!
!1606R04_1606R06
KOLLISION_ZONE 6\Anfrage;
!
!1606R04_1606R06
KOLLISION_ZONE 7\Anfrage;
!
!1606R04_1606R06
KOLLISION_ZONE 8\Anfrage;
!
MoveJ LHP_600, vSchnell, fine, nomtcp1\WObj:=BS_1606_1A;
!
!1606R04_1606R06
KOLLISION_ZONE 1\Anfrage;
!
MoveJ LHP_005,vSchnell,z100,nomtcp1\WObj:=BS_1606_1A;
MoveJ LHP_010,vSchnell,z100,nomtcp1\WObj:=BS_1606_1A;
MoveJ LHP_015,vSchnell,z100,nomtcp1\WObj:=BS_1606_1A;
MoveJ LHP_020,vSchnell,z100,nomtcp1\WObj:=BS_1606_1A;
MoveJ LHP_025,vSchnell,z100,nomtcp1\WObj:=BS_1606_1A;
MoveJ LHP_030,vSchnell,z100,nomtcp1\WObj:=BS_1606_1A;
MoveJ LHP_035, vSchnell, z100, nomtcp1\WObj:=BS_1606_1A;
!
SpotL G0216023682BP20\VFO:=210,vSpot,nomtcp1\WObj:=BS_1606_1A;
!
MoveJ LHP_040,vSchnell,z100,nomtcp1\WObj:=BS_1606_1A;
!
SpotL G0216190516BP20\VFO:=210,vSpot,nomtcp1\WObj:=BS_1606_1A;
!
MoveJ LHP_045,vSchnell,z100,nomtcp1\WObj:=BS_1606_1A;
!
SpotL G0216190518BP20\VFO:=210,vSpot,nomtcp1\WObj:=BS_1606_1A;
!
SpotL G0216190520BP20\VFO:=210,vSpot,nomtcp1\WObj:=BS_1606_1A;
!
MoveJ LHP_050,vSchnell,z100,nomtcp1\WObj:=BS_1606_1A;
!
SpotL G0216190522BP20\VFO:=210,vSpot,nomtcp1\WObj:=BS_1606_1A;
!
SpotL G0216190524BP20\VFO:=210,vSpot,nomtcp1\WObj:=BS_1606_1A;
!
!1606R04_1606R03
KOLLISION_ZONE 4\Anfrage;
!
SpotL G0216190526BP20\VFO:=210,vSpot,nomtcp1\WObj:=BS_1606_1A;
!
SpotL G0216190528BP20\VFO:=210\Vorhub_Auf, vSpot, nomtcp1\WObj:=BS_1606_1A;
!
MoveJ LHP_055,vSchnell,z100,nomtcp1\WObj:=BS_1606_1A;
MoveJ LHP_060,vSchnell,z100,nomtcp1\WObj:=BS_1606_1A;
MoveJ LHP_065,vSchnell,z100,nomtcp1\WObj:=BS_1606_1A;
MoveJ LHP_070,vSchnell,z100,nomtcp1\WObj:=BS_1606_1A;
MoveJ LHP_075,vSchnell,z100,nomtcp1\WObj:=BS_1606_1A;
MoveJ LHP_080,vSchnell,z100,nomtcp1\WObj:=BS_1606_1A;
!
SpotL G0216190508BP20\VFO:=210,vSpot,nomtcp1\WObj:=BS_1606_1A;
!
MoveJ LHP_085,vSchnell,z100,nomtcp1\WObj:=BS_1606_1A;
MoveJ LHP_090,vSchnell,z100,nomtcp1\WObj:=BS_1606_1A;
!
SpotL G0216190506BP20\VFO:=210, vSpot, nomtcp1\WObj:=BS_1606_1A;
!
!1606R04_1606R03
KOLLISION_ZONE 4\Freigabe;
!
MoveJ LHP_205,vSchnell,z100,nomtcp1\WObj:=BS_1606_1A;
!
SpotL G0216023686BP20\VFO:=210, vSpot, nomtcp1\WObj:=BS_1606_1A;
!
SpotL G0216023688BP20\VFO:=210, vSpot, nomtcp1\WObj:=BS_1606_1A;
!
SpotL G0216190502BP20\VFO:=210\Vorhub_Auf, vSpot, nomtcp1\WObj:=BS_1606_1A;
!
MoveJ LHP_215, vSchnell, z100, nomtcp1\WObj:=BS_1606_1A;
MoveJ LHP_220, vSchnell, z100, nomtcp1\WObj:=BS_1606_1A;
!
!
SpotL G0213195684BP20\VFO:=210\Vorhub_Auf, vSpot, nomtcp1\WObj:=BS_1606_1A;
!
MoveJ LHP_225, vSchnell, z100, nomtcp1\WObj:=BS_1606_1A;
MoveJ LHP_230,vSchnell,z100,nomtcp1\WObj:=BS_1606_1A;
!
SpotL G0216190446BP20\VFO:=210\Vorhub_Auf,vSpot,nomtcp1\WObj:=BS_1606_1A;
!
MoveJ LHP_235,vSchnell,z100,nomtcp1\WObj:=BS_1606_1A;
MoveJ LHP_610, vSchnell, fine, nomtcp1\WObj:=BS_1606_1A;
!
!1606R04_1606R06
KOLLISION_ZONE 2\Anfrage;
!
MoveJ LHP_620,vSchnell,z100,nomtcp1\WObj:=BS_1606_1A;
MoveJ LHP_625,vSchnell,z100,nomtcp1\WObj:=BS_1606_1A;
!
SpotL G0216023684BP20\VFO:=210\Vorhub_Auf, vSpot, nomtcp1\WObj:=BS_1606_1A;
!
MoveJ LHP_630, vSchnell, z100, nomtcp1\WObj:=BS_1606_1A;
MoveJ LHP_635, vSchnell, z100, nomtcp1\WObj:=BS_1606_1A;
MoveJ LHP_645, vSchnell, z100, nomtcp1\WObj:=BS_1606_1A;
MoveJ LHP_115,vSchnell,z100,nomtcp1\WObj:=BS_1606_1A;
MoveJ LHP_120,vSchnell,z100,nomtcp1\WObj:=BS_1606_1A;
MoveJ LHP_125,vSchnell,z100,nomtcp1\WObj:=BS_1606_1A;
!
SpotL G0216190492BP20\VFO:=220\Vorhub_Auf,vSpot,nomtcp1\WObj:=BS_1606_1A;
!
MoveJ LHP_130,vSchnell,z100,nomtcp1\WObj:=BS_1606_1A;
MoveJ LHP_135,vSchnell,z1,nomtcp1\WObj:=BS_1606_1A;
MoveL LHP_140,vSchnell,z1,nomtcp1\WObj:=BS_1606_1A;
MoveL LHP_145,vSchnell,z1,nomtcp1\WObj:=BS_1606_1A;
!
SpotL G0216190582BP20\VFO:=210, vSpot, nomtcp1\WObj:=BS_1606_1A;
!
SpotL G0216190478BP20\VFO:=210\Vorhub_Auf,vSpot,nomtcp1\WObj:=BS_1606_1A;
!
MoveJ LHP_150,vSchnell,z1,nomtcp1\WObj:=BS_1606_1A;
MoveJ LHP_155,vSchnell,z1,nomtcp1\WObj:=BS_1606_1A;
MoveJ LHP_160,vSchnell,z1,nomtcp1\WObj:=BS_1606_1A;
MoveJ LHP_165,vSchnell,z100,nomtcp1\WObj:=BS_1606_1A;
MoveJ LHP_170,vSchnell,z100,nomtcp1\WObj:=BS_1606_1A;
MoveJ LHP_175,vSchnell,z100,nomtcp1\WObj:=BS_1606_1A;
MoveJ LHP_180, vSchnell, z100, nomtcp1\WObj:=BS_1606_1A;
!
!1606R04_1606R06
KOLLISION_ZONE 2\Freigabe;
!
MoveJ LHP_250, vSchnell, fine, nomtcp1\WObj:=BS_1606_1A;
!1606R04_1606R06
KOLLISION_ZONE 5\Anfrage;
!
MoveJ LHP_255,vSchnell,z100,nomtcp1\WObj:=BS_1606_1A;
MoveJ LHP_260,vSchnell,z100,nomtcp1\WObj:=BS_1606_1A;
MoveJ LHP_265,vSchnell,z100,nomtcp1\WObj:=BS_1606_1A;
MoveJ LHP_270,vSchnell,z100,nomtcp1\WObj:=BS_1606_1A;
MoveJ LHP_275,vSchnell,z100,nomtcp1\WObj:=BS_1606_1A;
MoveJ LHP_280, vSchnell, z100, nomtcp1\WObj:=BS_1606_1A;
MoveL LHP_285,vSchnell,z5,nomtcp1\WObj:=BS_1606_1A;
MoveL LHP_290,vSchnell,z5,nomtcp1\WObj:=BS_1606_1A;
MoveL LHP_295,vSchnell,z5,nomtcp1\WObj:=BS_1606_1A;
MoveL LHP_300,vSchnell,z5,nomtcp1\WObj:=BS_1606_1A;
MoveL LHP_305,vSchnell,z5,nomtcp1\WObj:=BS_1606_1A;
!
SpotL G0216190480BP20\VFO:=210\Vorhub_Auf, vSpot, nomtcp1\WObj:=BS_1606_1A;
!
MoveL LHP_310,vSchnell,z5,nomtcp1\WObj:=BS_1606_1A;
MoveL LHP_315,vSchnell,z5,nomtcp1\WObj:=BS_1606_1A;
MoveL LHP_320,vSchnell,z5,nomtcp1\WObj:=BS_1606_1A;
MoveL LHP_325,vSchnell,z5,nomtcp1\WObj:=BS_1606_1A;
MoveL LHP_330,vSchnell,z5,nomtcp1\WObj:=BS_1606_1A;
MoveL LHP_335,vSchnell,z5,nomtcp1\WObj:=BS_1606_1A;
MoveL LHP_340,vSchnell,z5,nomtcp1\WObj:=BS_1606_1A;
!
SpotL G0216022394BP20\VFO:=220\Vorhub_Auf,vSpot,nomtcp1\WObj:=BS_1606_1A;
!
MoveJ LHP_345, vSchnell, fine, nomtcp1\WObj:=BS_1606_1A;
!
!1606R04_1606R06
KOLLISION_ZONE 6\Freigabe;
!
MoveJ LHP_350, vSchnell, z100, nomtcp1\WObj:=BS_1606_1A;
!
SpotL G0216022386BP20\VFO:=210, vSpot, nomtcp1\WObj:=BS_1606_1A;
!
SpotL G0216047033BP20\VFO:=210,vSpot,nomtcp1\WObj:=BS_1606_1A;
!
SpotL G0216047032BP20\VFO:=210\Vorhub_Auf, vSpot, nomtcp1\WObj:=BS_1606_1A;
!
MoveJ LHP_355,vSchnell,z100,nomtcp1\WObj:=BS_1606_1A;
MoveJ LHP_360,vSchnell,z100,nomtcp1\WObj:=BS_1606_1A;
MoveJ LHP_365, vSchnell, z100, nomtcp1\WObj:=BS_1606_1A;
MoveJ LHP_370, vSchnell, z100, nomtcp1\WObj:=BS_1606_1A;
MoveJ LHP_375, vSchnell, z100, nomtcp1\WObj:=BS_1606_1A;
MoveJ LHP_380, vSchnell, z100, nomtcp1\WObj:=BS_1606_1A;
MoveJ LHP_385, vSchnell, z100, nomtcp1\WObj:=BS_1606_1A;
MoveJ LHP_390, vSchnell, fine, nomtcp1\WObj:=BS_1606_1A;
!
!1606R04_1606R06
KOLLISION_ZONE 7\Freigabe;
!
SpotL G0216190494BP20\VFO:=210,vSpot,nomtcp1\WObj:=BS_1606_1A;
!
SpotL G0216190496BP20\VFO:=210,vSpot,nomtcp1\WObj:=BS_1606_1A;
!
SpotL G0216190498BP20\VFO:=210,vSpot,nomtcp1\WObj:=BS_1606_1A;
!
MoveJ LHP_395,vSchnell,z100,nomtcp1\WObj:=BS_1606_1A;
!
SpotL G0216190488BP20\VFO:=210,vSpot,nomtcp1\WObj:=BS_1606_1A;
!
MoveJ LHP_400,vSchnell,z100,nomtcp1\WObj:=BS_1606_1A;
!
SpotL G0216190500BP20\VFO:=210\Vorhub_Auf,vSpot,nomtcp1\WObj:=BS_1606_1A;
!
MoveJ LHP_405,vSchnell,z100,nomtcp1\WObj:=BS_1606_1A;
MoveJ LHP_410,vSchnell,z100,nomtcp1\WObj:=BS_1606_1A;
MoveJ LHP_415,vSchnell,z100,nomtcp1\WObj:=BS_1606_1A;
MoveJ LHP_420,vSchnell,z100,nomtcp1\WObj:=BS_1606_1A;
MoveJ LHP_425,vSchnell,z100,nomtcp1\WObj:=BS_1606_1A;
MoveJ LHP_430,vSchnell,z100,nomtcp1\WObj:=BS_1606_1A;
MoveJ LHP_435,vSchnell,z100,nomtcp1\WObj:=BS_1606_1A;
!
SpotL G0216047028BP20\VFO:=210,vSpot,nomtcp1\WObj:=BS_1606_1A;
!
SpotL G0216047029BP20\VFO:=210,vSpot,nomtcp1\WObj:=BS_1606_1A;
!
SpotL G0216022368BP20\VFO:=210,vSpot,nomtcp1\WObj:=BS_1606_1A;
!
SpotL G0216022370BP20\VFO:=210\Vorhub_Auf,vSpot,nomtcp1\WObj:=BS_1606_1A;
!
MoveJ LHP_440, vSchnell, z100, nomtcp1\WObj:=BS_1606_1A;
MoveJ LHP_445, vSchnell, z100, nomtcp1\WObj:=BS_1606_1A;
MoveJ LHP_450, vSchnell, z100, nomtcp1\WObj:=BS_1606_1A;
MoveJ LHP_455, vSchnell, z100, nomtcp1\WObj:=BS_1606_1A;
MoveJ LHP_460, vSchnell, z100, nomtcp1\WObj:=BS_1606_1A;
MoveJ LHP_465, vSchnell, z100, nomtcp1\WObj:=BS_1606_1A;
!
SpotL G0216190436BP20\VFO:=210,vSpot,nomtcp1\WObj:=BS_1606_1A;
!
SpotL G0216190438BP20\VFO:=210,vSpot,nomtcp1\WObj:=BS_1606_1A;
!
SpotL G0216190440BP20\VFO:=210, vSpot, nomtcp1\WObj:=BS_1606_1A;
!
SpotL G0216023676BP20\VFO:=210,vSpot,nomtcp1\WObj:=BS_1606_1A;
!
SpotL G0216023674BP20\VFO:=210,vSpot,nomtcp1\WObj:=BS_1606_1A;
!
MoveJ LHP_470, vSchnell, fine, nomtcp1\WObj:=BS_1606_1A;
!
!1606R04_1606R06
KOLLISION_ZONE 8\Freigabe;
!
SpotL G0216023672BP20\VFO:=210,vSpot,nomtcp1\WObj:=BS_1606_1A;
!
SpotL G0216023670BP20\VFO:=210,vSpot,nomtcp1\WObj:=BS_1606_1A;
!
SpotL G0213195682BP20\VFO:=210,vSpot,nomtcp1\WObj:=BS_1606_1A;
!
SpotL G0213195680BP20\VFO:=210,vSpot,nomtcp1\WObj:=BS_1606_1A;
!
SpotL G0216190428BP20\VFO:=210,vSpot,nomtcp1\WObj:=BS_1606_1A;
!
SpotL G0216190430BP20\VFO:=210,vSpot,nomtcp1\WObj:=BS_1606_1A;
!
SpotL G0216190432BP20\VFO:=210,vSpot,nomtcp1\WObj:=BS_1606_1A;
!
SpotL G0216190434BP20\VFO:=210\Vorhub_Auf, vSpot, nomtcp1\WObj:=BS_1606_1A;
!
MoveJ LHP_475,vSchnell,z100,nomtcp1\WObj:=BS_1606_1A;
MoveJ LHP_480, vSchnell, z100, nomtcp1\WObj:=BS_1606_1A;
!
!
SpotL G0216190576BP20\VFO:=220,vSpot,nomtcp1\WObj:=BS_1606_1A;
!
SpotL G0213195678BP20\VFO:=210\Vorhub_Auf,vSpot,nomtcp1\WObj:=BS_1606_1A;
!
MoveJ LHP_485,vSchnell,z100,nomtcp1\WObj:=BS_1606_1A;
MoveJ LHP_490,vSchnell,z100,nomtcp1\WObj:=BS_1606_1A;
!
SpotL G0213195686BP20\VFO:=210,vSpot,nomtcp1\WObj:=BS_1606_1A;
!
SpotL G0213195688BP20\VFO:=210\Vorhub_Auf, vSpot, nomtcp1\WObj:=BS_1606_1A;
!
MoveJ LHP_495, vSchnell, z100, nomtcp1\WObj:=BS_1606_1A;
MoveJ LHP_500, vSchnell, z10, nomtcp1\WObj:=BS_1606_1A;
MoveJ LHP_505, vSchnell, z5, nomtcp1\WObj:=BS_1606_1A;
MoveJ LHP_510, vSchnell, z5, nomtcp1\WObj:=BS_1606_1A;
MoveJ LHP_515, vSchnell, z5, nomtcp1\WObj:=BS_1606_1A;
MoveJ LHP_520, vSchnell, z5, nomtcp1\WObj:=BS_1606_1A;
MoveJ LHP_525, vSchnell, z5, nomtcp1\WObj:=BS_1606_1A;
MoveJ LHP_530, vSchnell, fine, nomtcp1\WObj:=BS_1606_1A;
!
!1606R04_1606R06
KOLLISION_ZONE 1\Freigabe;
!
MoveJ LHP_535, vSchnell, z100, nomtcp1\WObj:=BS_1606_1A;
!
MoveJ ToolHome1,vSchnell,fine,nomtcp1;
!
!1606R04_1606R06
KOLLISION_ZONE 5\Freigabe;
!
ABL 254\ABL_WAIT;
ABL 255\ABL_SET;
!
!1606R04_1606R06
KOLLISION_ZONE 9\Anfrage;
!
!1606R04_1606R06
KOLLISION_ZONE 9\Freigabe;
!
ENDPROC




ENDMODULE
